FUNCTION_BLOCK FB_Base
VAR_INPUT
	Input1 : INT;
	Input2 : REAL;
END_VAR
VAR_OUTPUT
	Output1 : DINT;
	Output2 : LREAL;
END_VAR
VAR
	Internal1 : SINT;
	Internal2 : WORD;
	Internal3 : ST_Complex_1;
END_VAR

END_FUNCTION_BLOCK

(* stored: Version 1.1.0.1, ProductVersion 3.1.4024.0
   POU FB_Base: Id {653ed6c8-6e1e-486f-ad95-85cd0ad84f7e}, SpecialFunc None *)
